FUNCTION_BLOCK RT_E_PERMIT (* Permissive propagation of an event *)
  (* Version 1.0, 2008-07-10, Alois Zoitl, ACIN *)
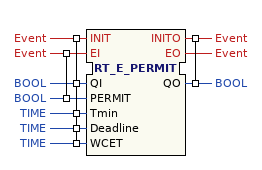
  EVENT_INPUT
    INIT WITH QI, Tmin, Deadline, WCET;
    EI WITH PERMIT; (* Event input *)
  END_EVENT
  EVENT_OUTPUT
    INITO WITH QO;
    EO; (* Event output *)
  END_EVENT
  VAR_INPUT
    QI : BOOL;
    PERMIT : BOOL;
    Tmin : TIME;
    Deadline : TIME;
    WCET : TIME;
  END_VAR
  VAR_OUTPUT
    QO : BOOL;
  END_VAR
END_FUNCTION_BLOCK
(* other elements stored in the file *)
(* Identificatiovn Description=Copyright (c) 2008 ACIN This program and the accompanying materials are made available under the terms of the Eclipse Public License 2.0 which is available at https://www.eclipse.org/legal/epl-2.0/ SPDX-License-Identifier: EPL-2.0 *)
